// TIA Portal V14 SP1 export
// export: Created 2020-10-16T18:41:45.2536874Z, ExportSetting None, DisplayName Totally Integrated Automation Portal, DisplayVersion V14 SP1 Update 3, DisplayName TIA Portal Openness, DisplayVersion V14 SP1 Update 2, DisplayName SINAMICS Startdrive, DisplayVersion V14 SP1 Update 4, DisplayName STEP 7 Professional, DisplayVersion V14 SP1 Update 3, DisplayName STEP 7 Safety, DisplayVersion V14 SP1, DisplayName WinCC Professional, DisplayVersion V14 SP1 Update 3, DisplayName SIMATIC Visualization Architect, DisplayVersion V14 SP1 Update 3
FUNCTION_BLOCK "FB_SEQ_One"   // FB1234, GRAPH
{ S7_Optimized_Access := 'TRUE' }
// stored: GraphVersion 4.0, InitialValuesAcquisition false, SetENOAutomatically false
   // inherited from GRAPH_BASE
   VAR_INPUT
      OFF_SQ { ExternalAccessible := 'False'; ExternalVisible := 'False'; ExternalWritable := 'False'} : Bool := false;   // Kette ausschalten
      INIT_SQ { ExternalAccessible := 'False'; ExternalVisible := 'False'; ExternalWritable := 'False'} : Bool := false;   // Kette in Initialzustand versetzen
      ACK_EF { ExternalAccessible := 'False'; ExternalVisible := 'False'; ExternalWritable := 'False'} : Bool := false;   // Alle Fehler und Störungen quittieren
      S_PREV { ExternalAccessible := 'False'; ExternalVisible := 'False'; ExternalWritable := 'False'} : Bool := false;   // Vorherigen Schritt am Parameter S_NO ausgeben
      S_NEXT { ExternalAccessible := 'False'; ExternalVisible := 'False'; ExternalWritable := 'False'} : Bool := false;   // Nächsten Schritt am Parameter S_NO anzeigen
      SW_AUTO { ExternalAccessible := 'False'; ExternalVisible := 'False'; ExternalWritable := 'False'} : Bool := false;   // Automatischer Betrieb
      SW_TAP { ExternalAccessible := 'False'; ExternalVisible := 'False'; ExternalWritable := 'False'} : Bool := false;   // Halbautomatisch/Weiterschalten mit Transition
      SW_TOP { ExternalAccessible := 'False'; ExternalVisible := 'False'; ExternalWritable := 'False'} : Bool := false;   // Halbautomatisch/Ignoriere Transition
      SW_MAN { ExternalAccessible := 'False'; ExternalVisible := 'False'; ExternalWritable := 'False'} : Bool := false;   // Handbetrieb
      S_SEL { ExternalAccessible := 'False'; ExternalVisible := 'False'; ExternalWritable := 'False'} : Int := 0;   // Schritt auswählen, der an S_NO ausgegeben werden soll
      S_ON { ExternalAccessible := 'False'; ExternalVisible := 'False'; ExternalWritable := 'False'} : Bool := false;   // Schritt aktivieren, der an Parameter S_NO anliegt
      S_OFF { ExternalAccessible := 'False'; ExternalVisible := 'False'; ExternalWritable := 'False'} : Bool := false;   // Schritt deaktivieren, der an Parameter S_NO anliegt
      T_PUSH { ExternalAccessible := 'False'; ExternalVisible := 'False'; ExternalWritable := 'False'} : Bool := false;   // Schaltfreigabe für Transition im halbautomatischen Betrieb
   END_VAR
   VAR_OUTPUT
      S_NO { ExternalAccessible := 'False'; ExternalVisible := 'False'; ExternalWritable := 'False'} : Int := 0;   // Schrittnummer
      S_MORE { ExternalAccessible := 'False'; ExternalVisible := 'False'; ExternalWritable := 'False'} : Bool := false;   // Weitere Schritte sind vorhanden und können in S_NO angezeigt werden.
      S_ACTIVE { ExternalAccessible := 'False'; ExternalVisible := 'False'; ExternalWritable := 'False'} : Bool := false;   // Schritt, der an Parameter S_NO angezeigt wird, ist aktiv
      ERR_FLT { ExternalAccessible := 'False'; ExternalVisible := 'False'; ExternalWritable := 'False'} : Bool := false;   // Sammelfehler Interlock oder Supervision
      AUTO_ON { ExternalAccessible := 'False'; ExternalVisible := 'False'; ExternalWritable := 'False'} : Bool := false;   // Automatischer Betrieb eingeschaltet
      TAP_ON { ExternalAccessible := 'False'; ExternalVisible := 'False'; ExternalWritable := 'False'} : Bool := false;   // Halbautomatischer Betrieb/Schritt mit Transition eingeschaltet
      TOP_ON { ExternalAccessible := 'False'; ExternalVisible := 'False'; ExternalWritable := 'False'} : Bool := false;   // Halbautomatischer Betrieb/Ignoriere Transition eingeschaltet
      MAN_ON { ExternalAccessible := 'False'; ExternalVisible := 'False'; ExternalWritable := 'False'} : Bool := false;   // Handbetrieb eingeschaltet
   END_VAR
   VAR
      "NextStep (1)" { ExternalAccessible := 'False'; ExternalVisible := 'False'; ExternalWritable := 'False'} : G7_TransitionPlus_V4;   // Transitionsstruktur
      "NextStep (21)" { ExternalAccessible := 'False'; ExternalVisible := 'False'; ExternalWritable := 'False'} : G7_TransitionPlus_V4;   // Transitionsstruktur
      "AbortStep (121)" { ExternalAccessible := 'False'; ExternalVisible := 'False'; ExternalWritable := 'False'} : G7_TransitionPlus_V4;   // Transitionsstruktur
      "OptionStep (221)" { ExternalAccessible := 'False'; ExternalVisible := 'False'; ExternalWritable := 'False'} : G7_TransitionPlus_V4;   // Transitionsstruktur
      "NextStep (27)" { ExternalAccessible := 'False'; ExternalVisible := 'False'; ExternalWritable := 'False'} : G7_TransitionPlus_V4;   // Transitionsstruktur
      "NextStep (32)" { ExternalAccessible := 'False'; ExternalVisible := 'False'; ExternalWritable := 'False'} : G7_TransitionPlus_V4;   // Transitionsstruktur
      "NextStep (43)" { ExternalAccessible := 'False'; ExternalVisible := 'False'; ExternalWritable := 'False'} : G7_TransitionPlus_V4;   // Transitionsstruktur
   END_VAR
BEGIN
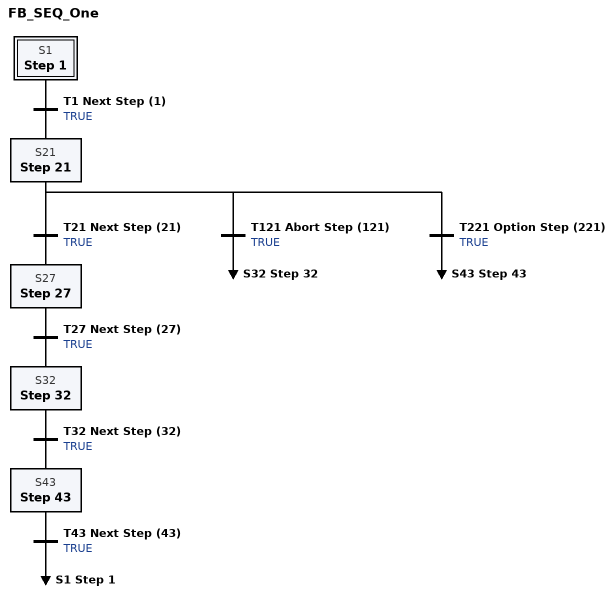
   // sequencer 1: My step sequence
   // My step sequecne comment
   INITIAL_STEP "Step 1":   // S1, max time T#10S, warning time T#7S
      // Action Step 1
   END_STEP
   TRANSITION "Next Step (1)" FROM "Step 1" TO "Step 21"   // T1
      := TRUE;
   END_TRANSITION
   STEP "Step 21":   // S21, max time T#10S, warning time T#7S
      // Action Step 21
   END_STEP
   TRANSITION "Next Step (21)" FROM "Step 21" TO "Step 27"   // T21
      := TRUE;
   END_TRANSITION
   TRANSITION "Abort Step (121)" FROM "Step 21" TO "Step 32"   // T121, jump
      := TRUE;
   END_TRANSITION
   TRANSITION "Option Step (221)" FROM "Step 21" TO "Step 43"   // T221, jump
      := TRUE;
   END_TRANSITION
   STEP "Step 27":   // S27, max time T#10S, warning time T#7S
      // Action Step 27
   END_STEP
   TRANSITION "Next Step (27)" FROM "Step 27" TO "Step 32"   // T27
      := TRUE;
   END_TRANSITION
   STEP "Step 32":   // S32, max time T#10S, warning time T#7S
      // Action Step 32
   END_STEP
   TRANSITION "Next Step (32)" FROM "Step 32" TO "Step 43"   // T32
      := TRUE;
   END_TRANSITION
   STEP "Step 43":   // S43, max time T#10S, warning time T#7S
      // Action Step 43
   END_STEP
   TRANSITION "Next Step (43)" FROM "Step 43" TO "Step 1"   // T43, jump
      := TRUE;
   END_TRANSITION
END_FUNCTION_BLOCK
